(*			
	EVERDE sp. z o.o.
	Rafał Osajda		08.08.2025		TC 4024.66
	Interfejs do wyciągania z SPM przez HMI danych do wyświetlania - dla ramki zmiana trybu
*)
INTERFACE ITF_SPM_HMI_04_Lacznik EXTENDS  B_Baza.ITF_ZrodloIdentyfikacji

METHOD PolaczZTablicamiZmianaTrybu : ST_SPM_HMI_04
END_METHOD

METHOD ZwrocZmianaTrybu : BOOL
VAR_INPUT
END_VAR
END_METHOD

END_INTERFACE

(* stored: Version 1.1.0.1
   Itf ITF_SPM_HMI_04_Lacznik: Id {17e3aea0-4cb8-0b8e-1baf-70aa0d9a9d22}
   Method PolaczZTablicamiZmianaTrybu: Id {de7cd170-f8df-0b26-0124-705ed73e491f}
   Method ZwrocZmianaTrybu: Id {c46eef9b-2703-0e2f-1c5b-eb098c3b66d0} *)
